// TIA Portal V20 export
DATA_BLOCK "Instance_FB_Marrige_DB"   // DB108
// stored: AutoNumber false, InstanceOfName FB_Marrige, InstanceOfType FB
"FB_Marrige"
   // VAR_INPUT
   //    In_Functional_Test_Odd : "IO_Device_Functinal_Test_Odd";
   //    In_Functional_Test_Even : "IO_Device_Functinal_Test_Even";
   //    Water_Fountain : String;
   //    Serial_Number : String[17];
   //    Read_Electrial_Voltage : UInt;
   // END_VAR
   // VAR_OUTPUT
   //    Functional_Tests_Panels : Array[0..31] of "Functional_Test";
   //    Got_Married : Bool;
   // END_VAR
   // VAR
   //    Aux_Trigger_0 : Bool;
   //    Aux_Trigger_1 : Bool;
   //    Aux_Trigger_2 : Bool;
   //    Aux_Trigger_3 : Bool;
   //    Aux_Trigger_4 : Bool;
   //    Aux_Trigger_5 : Bool;
   //    Aux_Trigger_6 : Bool;
   //    Aux_Trigger_7 : Bool;
   //    Aux_Trigger_8 : Bool;
   //    Aux_Trigger_9 : Bool;
   //    Aux_Trigger_10 : Bool;
   //    Aux_Trigger_11 : Bool;
   //    Aux_Trigger_12 : Bool;
   //    Aux_Trigger_13 : Bool;
   //    Aux_Trigger_14 : Bool;
   //    Aux_Trigger_15 : Bool;
   //    Aux_Trigger_16 : Bool;
   //    Aux_Trigger_17 : Bool;
   //    Aux_Trigger_18 : Bool;
   //    Aux_Trigger_19 : Bool;
   //    Aux_Trigger_20 : Bool;
   //    Aux_Trigger_21 : Bool;
   //    Aux_Trigger_22 : Bool;
   //    Aux_Trigger_23 : Bool;
   //    Aux_Trigger_24 : Bool;
   //    Aux_Trigger_25 : Bool;
   //    Aux_Trigger_26 : Bool;
   //    Aux_Trigger_27 : Bool;
   //    Aux_Trigger_28 : Bool;
   //    Aux_Trigger_29 : Bool;
   //    Aux_Trigger_30 : Bool;
   //    Aux_Trigger_31 : Bool;
   // END_VAR
BEGIN
END_DATA_BLOCK
